// TIA Portal project "SicaklikNem" (V19)

(* hardware
DEVICE "HMI_1"  MTP700 Unified Basic
   slot 0: "HMI_1"  MTP700 Unified Basic  6AV2 123-3GB32-0AW0  19.0.0.0
   slot 1: "HMI_RT_1"  MTP700 Unified Basic  6AV2 123-3GB32-0AW0  19.0.0.0
   slot 6: "HMI_1.IE_CP_1"  PROFINET Interface  19.0.0.0
      slot 1: "PROFINET Interface_GBit"  PROFINET Interface
         slot 1: "Port_1"  Port
DEVICE "S7-1200 station_1"  S7-1200 Station
   slot 0: "Rack_0"  S7-1200 Rack  Rack  V1.0
   slot 1: "PLC_1"  CPU 1211C DC/DC/DC  6ES7 211-1AE40-0XB0  V4.6
   slot 3: "CB 1241 (RS485)"  CB 1241 (RS485)  6ES7 241-1CH30-1XB0  V1.0
*)

// ===== PLC "PLC_1"  CPU 1211C DC/DC/DC =====

VAR_GLOBAL   // PLC tag table "Default tag table"
   "Clock_Byte" AT %MB0 : Byte;
   "Clock_10Hz" AT %M0.0 : Bool;
   "Clock_5Hz" AT %M0.1 : Bool;
   "Clock_2.5Hz" AT %M0.2 : Bool;
   "Clock_2Hz" AT %M0.3 : Bool;
   "Clock_1.25Hz" AT %M0.4 : Bool;
   "Clock_1Hz" AT %M0.5 : Bool;
   "Clock_0.625Hz" AT %M0.6 : Bool;
   "Clock_0.5Hz" AT %M0.7 : Bool;
   "System_Byte" AT %MB1 : Byte;
   "FirstScan" AT %M1.0 : Bool;
   "DiagStatusUpdate" AT %M1.1 : Bool;
   "AlwaysTRUE" AT %M1.2 : Bool;
   "AlwaysFALSE" AT %M1.3 : Bool;
   "mbDataAddr" AT %MD2 : UDInt;
   "mbAddr" AT %MW6 : UInt;
   "mbReq" AT %M8.0 : Bool;
   "mbMode" AT %MB9 : USInt;
   "mbDataLen" AT %MW10 : UInt;
   "iCounter" AT %MW12 : Int;
   "Tag_1" AT %MW500 : Int;
   "Tag_2" AT %MW502 : Int;
END_VAR

DATA_BLOCK "DB_Trig"   // DB1
{ S7_Optimized_Access := 'TRUE' }
VERSION : 0.1
   VAR
      "1" : Bool;
      "2" : Bool;
      "3" : Bool;
      "4" : Bool;
      "5" : Bool;
      "6" : Bool;
      "7" : Bool;
      "8" : Bool;
      "9" : Bool;
      "10" : Bool;
      "11" : Bool;
      "12" : Bool;
      "13" : Bool;
      "14" : Bool;
      "15" : Bool;
      "16" : Bool;
      "17" : Bool;
      "18" : Bool;
      "19" : Bool;
      "20" : Bool;
   END_VAR
BEGIN
END_DATA_BLOCK

FUNCTION "FC_Modbus" : Void   // FC1, LAD
{ S7_Optimized_Access := 'TRUE' }
VERSION : 0.1
   VAR_TEMP   // added for the SCL form of the ladder/FBD networks
      _w1 : Bool;
   END_VAR
BEGIN

REGION Network 1
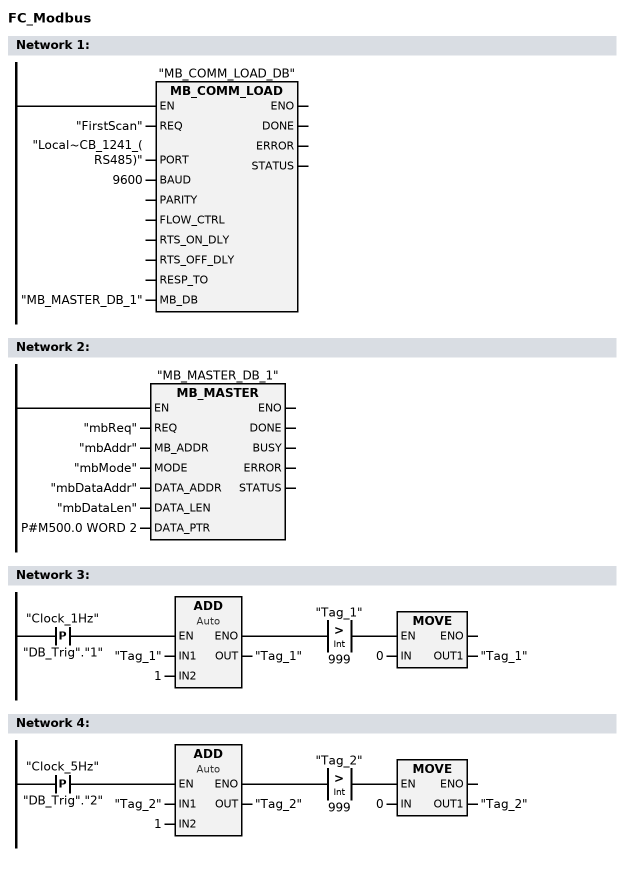
   "MB_COMM_LOAD_DB"(REQ := "FirstScan",   // MB_COMM_LOAD
                     PORT := "Local~CB_1241_(RS485)",
                     BAUD := 9600,
                     MB_DB := "MB_MASTER_DB_1");
END_REGION

REGION Network 2
   "MB_MASTER_DB_1"(REQ := "mbReq",   // MB_MASTER
                    MB_ADDR := "mbAddr",
                    MODE := "mbMode",
                    DATA_ADDR := "mbDataAddr",
                    DATA_LEN := "mbDataLen",
                    DATA_PTR := P#M500.0 WORD 2);
END_REGION

REGION Network 3
   RUNG wire#powerrail
      P_Contact(operand := "Clock_1Hz", bit := "DB_Trig"."1")
      Add(in1 := "Tag_1", in2 := 1, out => "Tag_1")
      { S7_Templates := "SrcType := Int" } GT_Contact(in1 := "Tag_1", in2 := 999)
      Move(in := 0, out1 => "Tag_1")
   END_RUNG
   // the same network as SCL:
   #_w1 := "Clock_1Hz" AND NOT "DB_Trig"."1";   // rising edge of "Clock_1Hz"
   "DB_Trig"."1" := "Clock_1Hz";
   IF #_w1 THEN "Tag_1" := "Tag_1" + 1; END_IF;
   IF #_w1 AND ("Tag_1" > 999) THEN "Tag_1" := 0; END_IF;
END_REGION

REGION Network 4
   RUNG wire#powerrail
      P_Contact(operand := "Clock_5Hz", bit := "DB_Trig"."2")
      Add(in1 := "Tag_2", in2 := 1, out => "Tag_2")
      { S7_Templates := "SrcType := Int" } GT_Contact(in1 := "Tag_2", in2 := 999)
      Move(in := 0, out1 => "Tag_2")
   END_RUNG
   // the same network as SCL:
   #_w1 := "Clock_5Hz" AND NOT "DB_Trig"."2";   // rising edge of "Clock_5Hz"
   "DB_Trig"."2" := "Clock_5Hz";
   IF #_w1 THEN "Tag_2" := "Tag_2" + 1; END_IF;
   IF #_w1 AND ("Tag_2" > 999) THEN "Tag_2" := 0; END_IF;
END_REGION
END_FUNCTION

ORGANIZATION_BLOCK "Main"   // OB1, LAD, ProgramCycle
TITLE = "Main Program Sweep (Cycle)"
{ S7_Optimized_Access := 'TRUE' }
VERSION : 0.1
   VAR_INPUT
      Initial_Call : Bool;   // Initial call of this OB
      Remanence : Bool;   // =True, if remanent data are available
   END_VAR
BEGIN

REGION Network 1
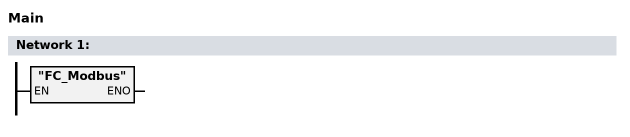
   RUNG wire#powerrail
      "FC_Modbus"()
   END_RUNG
   // the same network as SCL:
   "FC_Modbus"();
END_REGION
END_ORGANIZATION_BLOCK

(* ===== HMI "HMI_RT_1" =====
connection "Connection_1": ETHERNET, ILRT_S7_1500_OMS

text list "SystemTextList_ConfigErrorAlarmTextLibrary_1": 1 'NameService configuration error: Implicit deletion. Subelement instance @6%s@ must be deleted explicitly.'; 2 'NameService configuration error: Implicit deletion. Alias/Format/Unit instance @6%s@ must be deleted explicitly.'

text list "SystemTextList_ConfigErrorAlarmTextLibrary_2": 1 'EvDpManager::cleanupDeletedDatapoint - alert handler config is deleted implicitly for deleted datapoint, @3%s@'; 2 'EvDpManager::cleanupDeletedDatapoint - alert handler config is deleted implicitly but still has overrides, @3%s@'; 3 'EvDpManager::cleanupDeletedDatapoint - default value config is deleted implicitly for deleted datapoint, @3%s@'; 4 'EvDpManager::cleanupDeletedDatapoint - default value config is deleted implicitly but still has overrides, @3%s@'; 5 'EvDpManager::cleanupDeletedDatapoint - initial value config is deleted implicitly for deleted datapoint, @3%s@'; 6 'EvDpManager::cleanupDeletedDatapoint - initial value config is deleted implicitly but still has overrides, @3%s@'; 7 'EvDpManager::cleanupDeletedDatapoint - distribution config is deleted implicitly for deleted datapoint, @3%s@'; 8 'EvDpManager::cleanupDeletedDatapoint - distribution config is deleted implicitly but still has overrides, @3%s@'; 9 'EvDpManager::cleanupDeletedDatapoint - rangeCheck config is deleted implicitly for deleted datapoint, @3%s@'; 10 'EvDpManager::cleanupDeletedDatapoint - rangeCheck config is deleted implicitly but still has overrides, @3%s@'

text list "SystemTextList_ConfigErrorAlarmTextLibrary_3": 1 'The configured data point type was deleted, but a configured type is still defined for the node type: @3%s@.'; 2 'The configured data point node type was deleted in the data point type, but a configured type is still defined for the element: @3%s@.'

text list "SystemTextList_ConfigErrorAlarmTextLibrary_4": 2 'Cycles: @6%s@ does not exist'; 3 'Alarms: @6%s@ exists already'; 4 'Tags: Address @6%s@ was rejected'; 1 'Connections: @6%s@ does not exist'; 5 'Tags: Acquisition mode @6%s@ is not supported.'; 6 'Cycles: @6%s@ was deleted but associated tags exist.'; 7 'Connections: @6%s@ was deleted but associated tags exist.'; 8 'Tags: Tag @6%s@ was rejected.'; 9 'Tags: Tag @6%s@ has an invalid value.'; 0 'Connections: Connection to @6%s@ could not be established.'; 65638 'Connections: Connection to @6%s@ could not be established.'; 65639 'Connections: @6%s@ disconnected.'; 65640 'Connections: Connection to the HMI device @6%s@ is lost.'; 65641 'Connections: Connection to the PLC @6%s@ is lost.'; 65541 'Connections: Timeout while establishing the connection to @6%s@.'; 65542 'Connections: @6%s@ faulty.'; 65543 'Connections: Connection to the HMI device disconnected. Connection @5%s@ was changed.'; 65544 'Connections: Connection to the HMI device disconnected. Driver property was changed for connection @5%s@.'

text list "SystemTextList_ConfigErrorAlarmTextLibrary_5": 1 'Connections: Lifecycle monitoring cycle must be shorter than the response time.'; 2 'Connections: Cyclic services are configured but not supported by the target device.'; 3 'Connections: Change-controlled reading is configured but not supported by the target device.'; 4 'Tags: The address @6%s@ does not exist in the PLC.'; 5 'Tags: The default conversion type for the address @6%s@ could not be determined.'; 6 'Tags: Invalid conversion type'; 7 'Cycles: Invalid conversion type. Conversion is not supported at HmiCycle.'; 4096 'Connections: Version of the address @6%s@ is not supported.'; 4097 'Connections: PROFIBUS address is not supported.'; 4098 'Connections: Softbus address is not supported.'; 4099 'Connections: Address type @6%s@ is not supported.'; 4100 'Connections: Invalid connection name @6%s@. Access point is being ignored.'; 4101 'Connections: Routing is not supported. @6%s@ is not used.'; 4102 'Connections: Routing is not supported. @6%s@ is not used.'; 4103 'Connections: Invalid IP address @6%s@'; 4104 'Connections: Invalid Named Connection @6%s@. Valid format: >VMD</>connection<'; 4105 'Connections: Invalid Named Connection @6%s@. VMD connection name is too long. Only 24 characters are permitted.'; 4106 'Connections: Invalid Named Connection @6%s@. Connection name is too long. Only 32 characters are permitted.'; 4107 'Connections: Rack number @6%s@ is outside of the permitted range (0..7)'; 4108 'Connections: Invalid Named Connection @6%s@. Rack is ignored.'; 4109 'Connections: Slot number @6%s@ is outside of the permitted range (1..32)'; 4110 'Connections: Invalid Named Connection @6%s@. Slot is ignored.'; 4111 'Connection could not be established. Maximum number of available connections (@6%s@) has been exceeded.'; 4112 'Connection aborted. No sign of life in the last @4%s@ ms.'; 4113 'Connection could not be established - @4%s@'; 4114 'Connection could not be established. The address @6%s@ cannot be used.'; 4115 'Connection could not be established. Invalid address @6%s@'; 4116 'Connection could not be established - @4%s@'

text list "SystemTextList_ConfigErrorAlarmTextLibrary_6": 1 'Connection could not be established. Application instance certificate is not configured.'; 2 'Connection could not be established. Server has rejected the client certificate. OPC UA status code @4%s@.'; 3 'Connection could not be established. Internal problem in the certificate store. OPC UA status code @4%s@'; 4 'Connection could not be established. Application instance certificate could not be loaded. OPC UA status code @4%s@'; 5 'Connection could not be established. Server has not provided a certificate. @4%s@'; 6 'Connection could not be established. Validation of server certificate has failed. OPC UA status code @4%s@.'; 7 'Connection was closed. Error during alarm synchronization. OPC UA status code @4%s@.'; 8 'Connection was closed. Alarm/event subscription has failed. The number of operations on the server has been exceeded.'; 9 'Connection was closed. Alarm/event subscription has failed. The number of alarm/event subscriptions on the server has been exceeded.'; 10 'Connection could not be established. Server reports a license problem. OPC UA status code @4%s@.'; 11 'Connection could not be established. Maximum number of server sessions has been exceeded.'; 12 'Connection could not be established. Safety configuration is inconsistent. @4%s@'; 13 'Connection could not be established. The address @4%s@ cannot be used.'; 14 'Connection could not be established. OPC UA status code @4%s@'; 15 'Connection aborted. OPC UA server was stopped.'; 16 'Connection aborted. No sign of life in the last @4%s@ ms.'; 17 'Connection was closed. OPC UA server maintenance.'; 18 'Connection could not be established. Invalid configuration of the authentication mode - @4%s@'; 19 'Connection could not be established. User could not be authenticated. OPC UA status code @4%s@'; 20 'Connection could not be established. Server does not permit anonymous connection. OPC UA status code @4%s@'; 21 'Connection could not be established. Certificate problem: Error when writing the safety-relevant data to @4%s@.'; 22 'Connection could not be established. Certificate problem: Unexpected file in the folder @4%s@ cannot be removed.'; 23 'Connection could not be established. User could not be authenticated. No user or password configured.'; 24 'Connection could not be established. Unexpected length of the server certificate. @4%s@'; 25 'Connection could not be established. @4%s@ is empty.'; 26 'Connection could not be established. @4%s@ has an unexpected format.'; 27 'Connection could not be established. Server endpoints cannot be read. OPC UA status code @4%s@'; 28 'Connection could not be established. No server endpoints were found. @4%s@'; 29 'Connection could not be established. Application instance certificate could not be found.'; 30 'Connection could not be established. Unexpected format of the certificate @4%s@.'; 31 'Connection could not be established. Unexpected format of the certificate block list @4%s@.'; 32 'Connection could not be established. User could not be authenticated. An encryption detail is invalid. @4%s@'; 34 'Connection could not be established. - The configured non-transparent redundancy mode @4%s@ is not supported.'; 101 'Tags: Address @6%s@ does not exist on the server.'; 103 'Tags: Address @6%s@ cannot be accessed.'; 104 'Tags: Acquisition mode is not supported for address @6%s@.'; 201 'Alarms: Address @6%s@ does not exist on the server.'; 202 'Alarms: Address @6%s@ cannot be used. The specified range filter is not an OPC UA Event Notifier.'; 203 'Alarms: Address @6%s@ cannot be used. The specified range filter does not exist on the server.'; 204 'Alarms: Address @6%s@ cannot be used because it is not an OPC UA event type.'; 205 'Alarms: Address @6%s@ cannot be used because the OPC UA condition type is not supported.'; 206 'Alarms: Address @6%s@ cannot be used because the event type does not exist on the server.'; 207 'Alarms: Acquisition type cannot be used for address @6%s@.'; 301 'Address @6%s@ cannot be used because the version number is missing.'; 302 'Address @6%s@ cannot be used because the version number is invalid.'; 303 'Address @6%s@ cannot be used because the number of '$' delimiters is invalid.'; 304 'Address @6%s@ cannot be used because the address type is invalid.'; 305 'Unsupported version @6%s@ of the address'; 401 'Unexpected OPC UA server response: @6%s@'

text list "SystemTextList_ConfigErrorAlarmTextLibrary_7": 1 'Messages: Invalid condition string for the alarm view @6%s@.'; 2 'Messages: Invalid status tag and bit for the alarm view @6%s@.'; 3 'Messages: Invalid control tag and bit for the alarm view @6%s@.'

text list "SystemTextList_ConfigErrorAlarmTextLibrary_8": 1 'Logs: Implicit deletion. Logging tag instance @6%s@ should be deleted but there are overloaded elements.'

text list "SystemTextList_ConfigErrorAlarmTextLibrary_9": 1 ''; 2 'Restart of the runtime is required.'; 3 'The correct storage medium must be ejected and inserted again.'

text list "SystemTextList_ConfigErrorAlarmTextLibrary_10": 1 'CDS cache - Cache folder cannot be created or reached: @6%s@'; 2 'LOC cache - Cache folder cannot be created or reached: @6%s@'

text list "SystemTextList_RuntimeCollaborationFailureReason_1": 0 'Unknown error (@3%s@)'; 1 'The system is not running or there is a network problem'; 2 'Runtime is not started on the target device.'; 3 'The System ID does not match the expected System ID (@3%s@)'; 4 'The Collaboration name does not match the expected Collaboration name '@3%s@''; 5 'Wrong or unknown certificate'; 6 'Revoked certificate'; 7 'The time difference is too big.'; 8 'No common supported message version'; 9 'System ID (@3%s@) already exists'; 10 'System name (@3%s@) already exists'; 11 'ID/Name in local configuration for Runtime Collaboration already exists'

text list "SystemTextList_S7PlusAlarmTextListCollection_1": 4096 'Connections: Connection to the PLC @4%s@ is lost'; 4097 'Connections: Connection to the HMI device @4%s@ is lost'; 4098 'Connections: Maximum number of connections exceeded - @4%s@'; 4099 'Out of resources on PLC - @4%s@'; 4100 'Legitimation failed, invalid or missing password - @4%s@'; 4101 'Request to open the connection failed - @4%s@'; 4102 'Connections: Cannot connect to PLC - @4%s@'; 4103 'Request to open the connection could not be sent'; 4104 'General certificate error for PLC - @4%s@'; 4105 'PLC certificate expired for PLC - @4%s@'; 4106 'PLC certificate is revoked for PLC - @4%s@'; 4107 'PLC certificate is untrustworthy. Manual trust is possible for - @4%s@'; 4108 'PLC certificate is untrustworthy. Manual trust is not possible for - @4%s@'

text list "SystemTextList_AllenBradleyEIPAlarmTextListCollection_7": 4096 'Connection lost on PLC side - @5%s@'; 4097 'Connection lost on HMI side - @5%s@'; 4098 'Maximum number of connections exceeded - @5%s@'; 4099 'Out of resources on PLC - @5%s@'; 4100 'Legitimation failed, invalid or missing password - @5%s@'; 4101 'Open request failed - @5%s@'; 4102 'Cannot connect to PLC - @5%s@'; 4103 'Open request could not be sent'; 4104 'root certificate expired for - @5%s@'; 4105 'PLC certificate untrusted for - @5%s@'

text list "SystemTextList_OmronEIPAlarmTextListCollection_6": 4096 'Connection lost on PLC side - @5%s@'; 4097 'Connection lost on HMI side - @5%s@'; 4098 'Maximum number of connections exceeded - @5%s@'; 4099 'Out of resources on PLC - @5%s@'; 4100 'Legitimation failed, invalid or missing password - @5%s@'; 4101 'Open request failed - @5%s@'; 4102 'Cannot connect to PLC - @5%s@'; 4103 'Open request could not be sent'; 4104 'root certificate expired for - @5%s@'; 4105 'PLC certificate untrusted for - @5%s@'

text list "SystemTextList_StdModbusTCPAlarmTextListCollection_5": 4096 'Connections: Connection to the PLC @5%s@ is lost'; 4097 'Connections: Connection to the HMI device @5%s@ is lost'; 4098 'Connections: Maximum number of connections exceeded - @5%s@'; 4099 'Out of resources on PLC - @5%s@'; 4100 'Legitimation failed, invalid or missing password - @5%s@'; 4101 'Request to open the connection failed - @5%s@'; 4102 'Connections: Cannot connect to PLC - @5%s@'; 4103 'Request to open the connection could not be sent'; 4104 'General certificate error for PLC - @5%s@'; 4105 'PLC certificate expired for PLC - @5%s@'; 4106 'PLC certificate is revoked for PLC - @5%s@'; 4107 'PLC certificate is untrustworthy. Manual trust is possible for - @5%s@'; 4108 'PLC certificate is untrustworthy. Manual trust is not possible for - @5%s@'

text list "SystemTextList_MitsubishiMCAlarmTextListCollection_4": 4096 'Connection lost on PLC side - @5%s@'; 4097 'Connection lost on HMI side - @5%s@'; 4098 'Maximum number of connections exceeded - @5%s@'; 4099 'Out of resources on PLC - @5%s@'; 4100 'Legitimation failed, invalid or missing password - @5%s@'; 4101 'Open request failed - @5%s@'; 4102 'Cannot connect to PLC - @5%s@'; 4103 'Open request could not be sent'; 4104 'root certificate expired for - @5%s@'; 4105 'PLC certificate untrusted for - @5%s@'

text list "SystemTextList_MitsubishiiQAlarmTextListCollection_3": 4096 'Connection lost on PLC side - @5%s@'; 4097 'Connection lost on HMI side - @5%s@'; 4098 'Maximum number of connections exceeded - @5%s@'; 4099 'Out of resources on PLC - @5%s@'; 4100 'Legitimation failed, invalid or missing password - @5%s@'; 4101 'Open request failed - @5%s@'; 4102 'Cannot connect to PLC - @5%s@'; 4103 'Open request could not be sent'; 4104 'root certificate expired for - @5%s@'; 4105 'PLC certificate untrusted for - @5%s@'

text list "SystemTextList_StdModbusRTUAlarmTextListCollection_8": 4096 'Connections: Connection to the PLC @5%s@ is lost'; 4097 'Connections: Connection to the HMI device @5%s@ is lost'; 4098 'Connections: Maximum number of connections exceeded - @5%s@'; 4099 'Out of resources on PLC - @5%s@'; 4100 'Legitimation failed, invalid or missing password - @5%s@'; 4101 'Request to open the connection failed - @5%s@'; 4102 'Connections: Cannot connect to PLC - @5%s@'; 4103 'Request to open the connection could not be sent'; 4104 'General certificate error for PLC - @5%s@'; 4105 'PLC certificate expired for PLC - @5%s@'; 4106 'PLC certificate is revoked for PLC - @5%s@'; 4107 'PLC certificate is untrustworthy. Manual trust is possible for - @5%s@'; 4108 'PLC certificate is untrustworthy. Manual trust is not possible for - @5%s@'
*)